FUNCTION_BLOCK FB_LIGHT
VAR_INPUT

	ix_START: BOOL;
END_VAR
VAR_OUTPUT
	LIGHT: BOOL;
END_VAR
VAR
	STATE: INT;
	T_CYCLE: TON;
END_VAR

// --- CASE state machine ---
CASE STATE OF
    0: // Idle
        LIGHT := FALSE;
        // Stop cycle timer
        T_CYCLE(IN := FALSE);
        // Start cycle
        IF ix_START THEN
            STATE := 1;
        END_IF;
    1: // Start 30s cycle
        // Stop cycle if start button released
        IF ix_START = FALSE THEN
            STATE := 0;
        END_IF;
        // Start timer
        T_CYCLE(IN := TRUE, PT := T#30S);
        // Timed outputs
        LIGHT := TRUE;
        // LIGHT timing: ON at 10s, OFF at 25s
        IF (T_CYCLE.ET >= T#10S) AND (T_CYCLE.ET < T#25S) THEN
            LIGHT := TRUE;
        ELSE
            LIGHT := FALSE;
        END_IF;
        // End of cycle
        IF T_CYCLE.Q THEN
            STATE := 0;
        END_IF;
END_CASE;

END_FUNCTION_BLOCK

(* stored: Version 1.1.0.1, ProductVersion 3.1.4024.15
   POU FB_LIGHT: Id {82c01140-285c-41f9-a20d-0a6b127f89d7}, SpecialFunc None *)
